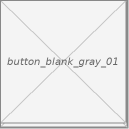
VISUALIZATION Blue_Ind  // 129x129
VAR_IN_OUT
	m_Input_Inst : None;
END_VAR
    Image (0,0 127x127), invisible if: (NOT m_Input_Inst) <> 0, image: button_blank_blue_01
    Image (0,0 126x123), invisible if: (m_Input_Inst) <> 0, image: button_blank_gray_01
END_VISUALIZATION

(* stored: Version 1.1.0.1, ProductVersion 3.1.4018.2
   Visu Blue_Ind: Id {84b70e07-2776-44bf-9aea-737f39653a92} *)
